TYPE ST_UN_CleanroomConnectSettings :
STRUCT
	stSettingsPalletConveyor : ST_SettingsPalletConveyor;
	stSettingsDockingInterface : ST_SettingsDockingInterface;
//##_LIFTING_TRANSPORT_DISABLED_##	stSettingsLiftingTransport : ST_SettingsLiftingTransport;
END_STRUCT
END_TYPE

(* stored: Version 1.1.0.1, ProductVersion 3.1.4024.12
   DUT ST_UN_CleanroomConnectSettings: Id {3f2f6cc8-3931-41b6-b35a-8f99944d8bca} *)
